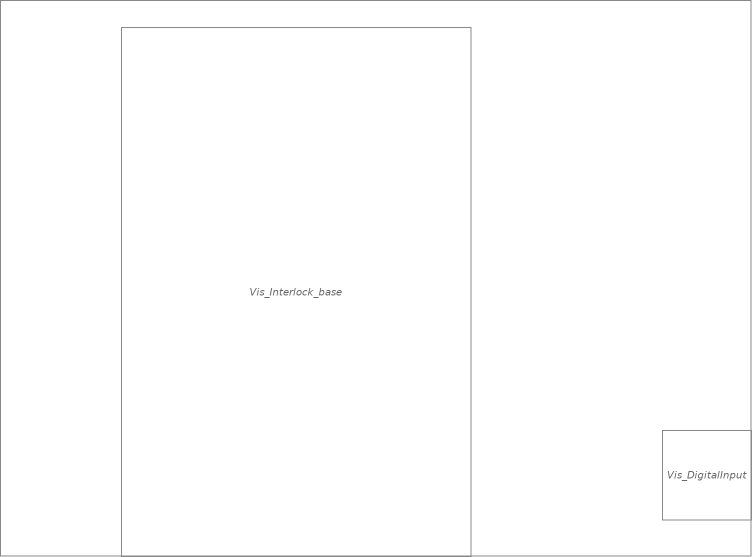
VISUALIZATION Visualization  // 752x557
    Frame (121,27 350x530)
        shows Vis_Interlock_base(stHMIInterlock := HMI.stTest01_Intlk)
    Frame (662,430 90x90)
        shows Vis_DigitalInput(stHMI_DigitalInput := HMI.stTest04_DigitalInput)
END_VISUALIZATION

(* stored: Version 1.1.0.1, ProductVersion 3.1.4024.11
   Visu Visualization: Id {b141f65d-7938-4a1a-903d-5d8a225011e6} *)
